// Mitsubishi GX Works2 project: 불켜기 예제1   PLC: Q03UDV

PROGRAM MAIN
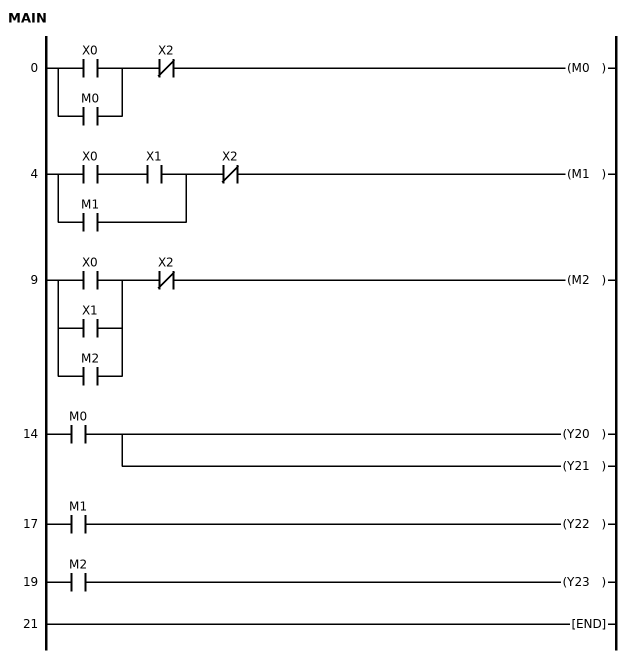
0     LD      X0
      OR      M0
      ANI     X2
      OUT     M0
4     LD      X0
      AND     X1
      OR      M1
      ANI     X2
      OUT     M1
9     LD      X0
      OR      X1
      OR      M2
      ANI     X2
      OUT     M2
14    LD      M0
      OUT     Y20
      OUT     Y21
17    LD      M1
      OUT     Y22
19    LD      M2
      OUT     Y23
21    END
END_PROGRAM
